FUNCTION_BLOCK HaltMover EXTENDS TaskBase
VAR_INPUT
END_VAR
VAR_OUTPUT
END_VAR
VAR
	haltMoverCA : Tc3_McCollisionAvoidance.MC_HaltCA;
	_Axis : REFERENCE TO Tc2_MC2.AXIS_REF;
	_HaltMover : BOOL;
END_VAR

{analysis -2}

METHOD Abort : BOOL
haltMoverCA.Execute := FALSE;
_Busy := FALSE;
_HaltMover := FALSE;
Abort := TRUE;
State := 0;
END_METHOD

METHOD Cycle : HRESULT
VAR_INPUT
END_VAR
Cycle := S_OK;
CASE State OF
	0:
		IF _HaltMover THEN
			Cycle := S_PENDING;
			_Done := FALSE;
			_Error := FALSE;
			_Busy := TRUE;
			haltMoverCA.Execute := TRUE;
			IF haltMoverCA.Busy THEN
				State := 10;
				_HaltMover := FALSE;
			END_IF
		END_IF
	
	10:
		IF NOT haltMoverCA.Busy THEN
			IF haltMoverCA.Done THEN
				_Done := TRUE;
			ELSIF haltMoverCA.Error THEN
				_Error := TRUE;
			END_IF
			_Busy := FALSE;
			haltMoverCA.Execute := FALSE;
			State := 0;
			Cycle := S_OK;
		END_IF
	ELSE
		Cycle := E_FAIL;
END_CASE

haltMoverCA(Axis := _Axis);
END_METHOD

PROPERTY Deceleration : MC_LREAL
GET
Deceleration := haltMoverCA.Deceleration;
END_GET
SET
haltMoverCA.Deceleration := Deceleration;
END_SET
END_PROPERTY

METHOD Execute : BOOL
VAR_INPUT
END_VAR
IF NOT _HaltMover THEN
	Execute := _HaltMover := TRUE;
ELSE
	Execute := false;
END_IF
END_METHOD

METHOD FB_init : BOOL
VAR_INPUT
	bInitRetains : BOOL; // if TRUE, the retain variables are initialized (warm start / cold start)
	bInCopyCode : BOOL;  // if TRUE, the instance afterwards gets moved into the copy code (online change)
	Axis : reference TO AXIS_REF;
END_VAR
_Axis REF= Axis;
END_METHOD

PROPERTY Gap : MC_LREAL
GET
Gap := haltMoverCA.Gap;
END_GET
SET
haltMoverCA.Gap := Gap;
END_SET
END_PROPERTY

PROPERTY Jerk : MC_LREAL
GET
Jerk := haltMoverCA.Jerk;
END_GET
SET
haltMoverCA.Jerk := Jerk;
END_SET
END_PROPERTY

END_FUNCTION_BLOCK

(* stored: Version 1.1.0.1
   POU HaltMover: Id {16fe934f-2b92-45c5-becd-cbf7a242dbb1}, SpecialFunc None
   Method Abort: Id {48a4c415-0254-4332-8d1a-2734e5dda505}
   Method Cycle: Id {1e7367c4-25b5-40fa-b219-770d9b7044ce}
   Property Deceleration: Id {c87d7270-1a2e-466f-a142-6139e2eda06f}
   Get Get: Id {a049ca93-b85d-4787-b520-72ad6ac74f0d}
   Set Set: Id {ae2611d3-59b2-4268-a7c2-500b25ff0ec0}
   Method Execute: Id {87eca2aa-365e-4c2f-b198-b62e8029fb82}
   Method FB_init: Id {0fd2927a-947b-415e-b53d-5482c2b0a045}
   Property Gap: Id {a94177ce-b18c-4479-ae6f-5707566b0317}
   Get Get: Id {ec2ed493-6955-4aef-baef-795d6fef3927}
   Set Set: Id {43b68502-e2f4-4b37-a3be-43a3ab3afcec}
   Property Jerk: Id {36146f01-bab8-49f7-9914-96e1977269b5}
   Get Get: Id {bd60b227-3eb3-44e9-be6f-0a525b541f10}
   Set Set: Id {356145f4-af65-48cf-aa74-d0bf709b5382} *)
